   cmCathodeNgPnp2ndFwdBwd.monitoring.commandWorkPos := FALSE;
   cmCathodeNgPnp2ndFwdBwd.monitoring.goToHomePos := TRUE;
   cmCathodeNgPnp2ndFwdBwd.monitoring.goToWorkPos := FALSE;
   cmCathodeNgPnp2ndFwdBwd.monitoring.inHomePos := TRUE;
   cmCathodeNgPnp2ndFwdBwd.monitoring.inWorkPos := FALSE;
   cmCathodeNgPnp2ndFwdBwd.monitoring.reset := FALSE;
   cmCathodeNgPnp2ndFwdBwd.monitoring.enableManualCmds := FALSE;
   cmCathodeNgPnp2ndFwdBwd.monitoring.error := FALSE;
   cmCathodeNgPnp2ndFwdBwd.monitoring.interlockHomePos := TRUE;
   cmCathodeNgPnp2ndFwdBwd.monitoring.interlockWorkPos := TRUE;
   cmCathodeNgPnp2ndFwdBwd.monitoring.status := 16#7004;
   cmCathodeNgPnp2ndFwdBwd.monitoring.interlockWarningWorkPos := FALSE;
   cmCathodeNgPnp2ndFwdBwd.monitoring.interlockWarningHomePos := FALSE;
   cmCathodeNgPnp2ndFwdBwd.configuration.referenceDesignator := WSTRING#'CaNgPnp2ndFwdBwd';
   cmCathodeNgPnp2ndFwdBwd.configuration.monitoringLeavingFeedback := T#5S;
   cmCathodeNgPnp2ndFwdBwd.configuration.monitoringReachingFeedback := T#5S;
   cmCathodeNgPnp2ndFwdBwd.configuration.monitoringDiscrepancy := T#0MS;
   cmCathodeNgPnp2ndFwdBwd.configuration.setOutputHomeContinuously := TRUE;
   cmCathodeNgPnp2ndFwdBwd.configuration.setOutputWorkContinuously := TRUE;
   cmCathodeNgPnp2ndFwdBwd.configuration.disableHomeCommand := FALSE;
   cmCathodeNgPnp2ndFwdBwd.configuration.disableFeedbackHomePos := FALSE;
   cmCathodeNgPnp2ndFwdBwd.configuration.disableFeedbackWorkPos := FALSE;
   cmCathodeNgPnp2ndFwdBwd.configuration.disableAlarms := FALSE;
   cmCathodeNgPnp2ndFwdBwd.configuration.resetOutputsOnError := FALSE;
   cmCathodeNgPnp2ndFwdBwd.configuration.allwaysWaitOnReachingTime := FALSE;
   cmCathodeMaintenanceMovingFixFrontRearFwdBwd.commands.refreshConfiguration := FALSE;
   cmCathodeMaintenanceMovingFixFrontRearFwdBwd.commands.editConfiguration := FALSE;
   cmCathodeMaintenanceMovingFixFrontRearFwdBwd.commands.saveConfiguration := FALSE;
   cmCathodeMaintenanceMovingFixFrontRearFwdBwd.commands.reset := FALSE;
   cmCathodeMaintenanceMovingFixFrontRearFwdBwd.commands.commandHomePos := FALSE;
   cmCathodeMaintenanceMovingFixFrontRearFwdBwd.commands.commandWorkPos := FALSE;
   cmCathodeMaintenanceMovingFixFrontRearFwdBwd.monitoring.enable := TRUE;
   cmCathodeMaintenanceMovingFixFrontRearFwdBwd.monitoring.referenceDesignator := WSTRING#'MaintenanceFix';
   cmCathodeMaintenanceMovingFixFrontRearFwdBwd.monitoring.commandHomePos := FALSE;
   cmCathodeMaintenanceMovingFixFrontRearFwdBwd.monitoring.commandWorkPos := FALSE;
   cmCathodeMaintenanceMovingFixFrontRearFwdBwd.monitoring.goToHomePos := FALSE;
   cmCathodeMaintenanceMovingFixFrontRearFwdBwd.monitoring.goToWorkPos := FALSE;
   cmCathodeMaintenanceMovingFixFrontRearFwdBwd.monitoring.inHomePos := FALSE;
   cmCathodeMaintenanceMovingFixFrontRearFwdBwd.monitoring.inWorkPos := FALSE;
   cmCathodeMaintenanceMovingFixFrontRearFwdBwd.monitoring.reset := FALSE;
   cmCathodeMaintenanceMovingFixFrontRearFwdBwd.monitoring.enableManualCmds := FALSE;
   cmCathodeMaintenanceMovingFixFrontRearFwdBwd.monitoring.error := FALSE;
   cmCathodeMaintenanceMovingFixFrontRearFwdBwd.monitoring.interlockHomePos := TRUE;
   cmCathodeMaintenanceMovingFixFrontRearFwdBwd.monitoring.interlockWorkPos := TRUE;
   cmCathodeMaintenanceMovingFixFrontRearFwdBwd.monitoring.status := 16#7003;
   cmCathodeMaintenanceMovingFixFrontRearFwdBwd.monitoring.interlockWarningWorkPos := FALSE;
   cmCathodeMaintenanceMovingFixFrontRearFwdBwd.monitoring.interlockWarningHomePos := FALSE;
   cmCathodeMaintenanceMovingFixFrontRearFwdBwd.configuration.referenceDesignator := WSTRING#'CaMaintFixFrontRearFwdBwd';
   cmCathodeMaintenanceMovingFixFrontRearFwdBwd.configuration.monitoringLeavingFeedback := T#5S;
   cmCathodeMaintenanceMovingFixFrontRearFwdBwd.configuration.monitoringReachingFeedback := T#5S;
   cmCathodeMaintenanceMovingFixFrontRearFwdBwd.configuration.monitoringDiscrepancy := T#0MS;
   cmCathodeMaintenanceMovingFixFrontRearFwdBwd.configuration.setOutputHomeContinuously := TRUE;
   cmCathodeMaintenanceMovingFixFrontRearFwdBwd.configuration.setOutputWorkContinuously := TRUE;
   cmCathodeMaintenanceMovingFixFrontRearFwdBwd.configuration.disableHomeCommand := FALSE;
   cmCathodeMaintenanceMovingFixFrontRearFwdBwd.configuration.disableFeedbackHomePos := FALSE;
   cmCathodeMaintenanceMovingFixFrontRearFwdBwd.configuration.disableFeedbackWorkPos := FALSE;
   cmCathodeMaintenanceMovingFixFrontRearFwdBwd.configuration.disableAlarms := FALSE;
   cmCathodeMaintenanceMovingFixFrontRearFwdBwd.configuration.resetOutputsOnError := FALSE;
   cmCathodeMaintenanceMovingFixFrontRearFwdBwd.configuration.allwaysWaitOnReachingTime := FALSE;
   cmCathodeNgBoxLiftUpDown.commands.refreshConfiguration := FALSE;
   cmCathodeNgBoxLiftUpDown.commands.editConfiguration := FALSE;
   cmCathodeNgBoxLiftUpDown.commands.saveConfiguration := FALSE;
   cmCathodeNgBoxLiftUpDown.commands.reset := FALSE;
   cmCathodeNgBoxLiftUpDown.commands.commandHomePos := FALSE;
   cmCathodeNgBoxLiftUpDown.commands.commandWorkPos := FALSE;
   cmCathodeNgBoxLiftUpDown.monitoring.enable := TRUE;
   cmCathodeNgBoxLiftUpDown.monitoring.referenceDesignator := WSTRING#'NgBoxLiftUpDown';
   cmCathodeNgBoxLiftUpDown.monitoring.commandHomePos := FALSE;
   cmCathodeNgBoxLiftUpDown.monitoring.commandWorkPos := FALSE;
   cmCathodeNgBoxLiftUpDown.monitoring.goToHomePos := FALSE;
   cmCathodeNgBoxLiftUpDown.monitoring.goToWorkPos := TRUE;
   cmCathodeNgBoxLiftUpDown.monitoring.inHomePos := FALSE;
   cmCathodeNgBoxLiftUpDown.monitoring.inWorkPos := TRUE;
   cmCathodeNgBoxLiftUpDown.monitoring.reset := FALSE;
   cmCathodeNgBoxLiftUpDown.monitoring.enableManualCmds := FALSE;
   cmCathodeNgBoxLiftUpDown.monitoring.error := FALSE;
   cmCathodeNgBoxLiftUpDown.monitoring.interlockHomePos := TRUE;
   cmCathodeNgBoxLiftUpDown.monitoring.interlockWorkPos := TRUE;
   cmCathodeNgBoxLiftUpDown.monitoring.status := 16#7006;
   cmCathodeNgBoxLiftUpDown.monitoring.interlockWarningWorkPos := FALSE;
   cmCathodeNgBoxLiftUpDown.monitoring.interlockWarningHomePos := FALSE;
   cmCathodeNgBoxLiftUpDown.configuration.referenceDesignator := WSTRING#'CaNgBoxLiftUpDown';
   cmCathodeNgBoxLiftUpDown.configuration.monitoringLeavingFeedback := T#5S;
   cmCathodeNgBoxLiftUpDown.configuration.monitoringReachingFeedback := T#5S;
   cmCathodeNgBoxLiftUpDown.configuration.monitoringDiscrepancy := T#0MS;
   cmCathodeNgBoxLiftUpDown.configuration.setOutputHomeContinuously := TRUE;
   cmCathodeNgBoxLiftUpDown.configuration.setOutputWorkContinuously := TRUE;
   cmCathodeNgBoxLiftUpDown.configuration.disableHomeCommand := FALSE;
   cmCathodeNgBoxLiftUpDown.configuration.disableFeedbackHomePos := FALSE;
   cmCathodeNgBoxLiftUpDown.configuration.disableFeedbackWorkPos := FALSE;
   cmCathodeNgBoxLiftUpDown.configuration.disableAlarms := FALSE;
   cmCathodeNgBoxLiftUpDown.configuration.resetOutputsOnError := FALSE;
   cmCathodeNgBoxLiftUpDown.configuration.allwaysWaitOnReachingTime := FALSE;
   cmCathodeNgBoxLockUpDown.commands.refreshConfiguration := FALSE;
   cmCathodeNgBoxLockUpDown.commands.editConfiguration := FALSE;
   cmCathodeNgBoxLockUpDown.commands.saveConfiguration := FALSE;
   cmCathodeNgBoxLockUpDown.commands.reset := FALSE;
   cmCathodeNgBoxLockUpDown.commands.commandHomePos := FALSE;
   cmCathodeNgBoxLockUpDown.commands.commandWorkPos := FALSE;
   cmCathodeNgBoxLockUpDown.monitoring.enable := TRUE;
   cmCathodeNgBoxLockUpDown.monitoring.referenceDesignator := WSTRING#'NgBoxLockUpDown';
   cmCathodeNgBoxLockUpDown.monitoring.commandHomePos := FALSE;
   cmCathodeNgBoxLockUpDown.monitoring.commandWorkPos := FALSE;
   cmCathodeNgBoxLockUpDown.monitoring.goToHomePos := FALSE;
   cmCathodeNgBoxLockUpDown.monitoring.goToWorkPos := FALSE;
   cmCathodeNgBoxLockUpDown.monitoring.inHomePos := FALSE;
   cmCathodeNgBoxLockUpDown.monitoring.inWorkPos := FALSE;
   cmCathodeNgBoxLockUpDown.monitoring.reset := FALSE;
   cmCathodeNgBoxLockUpDown.monitoring.enableManualCmds := FALSE;
   cmCathodeNgBoxLockUpDown.monitoring.error := FALSE;
   cmCathodeNgBoxLockUpDown.monitoring.interlockHomePos := TRUE;
   cmCathodeNgBoxLockUpDown.monitoring.interlockWorkPos := FALSE;
   cmCathodeNgBoxLockUpDown.monitoring.status := 16#7101;
   cmCathodeNgBoxLockUpDown.monitoring.interlockWarningWorkPos := FALSE;
   cmCathodeNgBoxLockUpDown.monitoring.interlockWarningHomePos := FALSE;
   cmCathodeNgBoxLockUpDown.configuration.referenceDesignator := WSTRING#'CaNgBoxLockUpDown';
   cmCathodeNgBoxLockUpDown.configuration.monitoringLeavingFeedback := T#5S;
   cmCathodeNgBoxLockUpDown.configuration.monitoringReachingFeedback := T#5S;
   cmCathodeNgBoxLockUpDown.configuration.monitoringDiscrepancy := T#0MS;
   cmCathodeNgBoxLockUpDown.configuration.setOutputHomeContinuously := TRUE;
   cmCathodeNgBoxLockUpDown.configuration.setOutputWorkContinuously := TRUE;
   cmCathodeNgBoxLockUpDown.configuration.disableHomeCommand := FALSE;
   cmCathodeNgBoxLockUpDown.configuration.disableFeedbackHomePos := FALSE;
   cmCathodeNgBoxLockUpDown.configuration.disableFeedbackWorkPos := FALSE;
   cmCathodeNgBoxLockUpDown.configuration.disableAlarms := FALSE;
   cmCathodeNgBoxLockUpDown.configuration.resetOutputsOnError := FALSE;
   cmCathodeNgBoxLockUpDown.configuration.allwaysWaitOnReachingTime := FALSE;
   cmCathodeNgPnpVaccum.commands.refreshConfiguration := FALSE;
   cmCathodeNgPnpVaccum.commands.editConfiguration := FALSE;
   cmCathodeNgPnpVaccum.commands.saveConfiguration := FALSE;
   cmCathodeNgPnpVaccum.commands.reset := FALSE;
   cmCathodeNgPnpVaccum.commands.commandHomePos := FALSE;
   cmCathodeNgPnpVaccum.commands.commandWorkPos := FALSE;
   cmCathodeNgPnpVaccum.monitoring.enable := TRUE;
   cmCathodeNgPnpVaccum.monitoring.referenceDesignator := WSTRING#'NgPnpVaccum';
   cmCathodeNgPnpVaccum.monitoring.commandHomePos := FALSE;
   cmCathodeNgPnpVaccum.monitoring.commandWorkPos := FALSE;
   cmCathodeNgPnpVaccum.monitoring.goToHomePos := FALSE;
   cmCathodeNgPnpVaccum.monitoring.goToWorkPos := FALSE;
   cmCathodeNgPnpVaccum.monitoring.inHomePos := TRUE;
   cmCathodeNgPnpVaccum.monitoring.inWorkPos := FALSE;
   cmCathodeNgPnpVaccum.monitoring.reset := FALSE;
   cmCathodeNgPnpVaccum.monitoring.enableManualCmds := FALSE;
   cmCathodeNgPnpVaccum.monitoring.error := FALSE;
   cmCathodeNgPnpVaccum.monitoring.interlockHomePos := TRUE;
   cmCathodeNgPnpVaccum.monitoring.interlockWorkPos := TRUE;
   cmCathodeNgPnpVaccum.monitoring.status := 16#7003;
   cmCathodeNgPnpVaccum.monitoring.interlockWarningWorkPos := FALSE;
   cmCathodeNgPnpVaccum.monitoring.interlockWarningHomePos := FALSE;
   cmCathodeNgPnpVaccum.configuration.referenceDesignator := WSTRING#'CaNgPnpVaccum';
   cmCathodeNgPnpVaccum.configuration.monitoringLeavingFeedback := T#5S;
   cmCathodeNgPnpVaccum.configuration.monitoringReachingFeedback := T#5S;
   cmCathodeNgPnpVaccum.configuration.monitoringDiscrepancy := T#0MS;
   cmCathodeNgPnpVaccum.configuration.setOutputHomeContinuously := TRUE;
   cmCathodeNgPnpVaccum.configuration.setOutputWorkContinuously := TRUE;
   cmCathodeNgPnpVaccum.configuration.disableHomeCommand := FALSE;
   cmCathodeNgPnpVaccum.configuration.disableFeedbackHomePos := FALSE;
   cmCathodeNgPnpVaccum.configuration.disableFeedbackWorkPos := FALSE;
   cmCathodeNgPnpVaccum.configuration.disableAlarms := FALSE;
   cmCathodeNgPnpVaccum.configuration.resetOutputsOnError := FALSE;
   cmCathodeNgPnpVaccum.configuration.allwaysWaitOnReachingTime := FALSE;
   cmCathodeConveyorCoverFwdBwd.commands.refreshConfiguration := FALSE;
   cmCathodeConveyorCoverFwdBwd.commands.editConfiguration := FALSE;
   cmCathodeConveyorCoverFwdBwd.commands.saveConfiguration := FALSE;
   cmCathodeConveyorCoverFwdBwd.commands.reset := FALSE;
   cmCathodeConveyorCoverFwdBwd.commands.commandHomePos := FALSE;
   cmCathodeConveyorCoverFwdBwd.commands.commandWorkPos := FALSE;
   cmCathodeConveyorCoverFwdBwd.monitoring.enable := TRUE;
   cmCathodeConveyorCoverFwdBwd.monitoring.referenceDesignator := WSTRING#'ConveyorCoverFwdBwd';
   cmCathodeConveyorCoverFwdBwd.monitoring.commandHomePos := FALSE;
   cmCathodeConveyorCoverFwdBwd.monitoring.commandWorkPos := FALSE;
   cmCathodeConveyorCoverFwdBwd.monitoring.goToHomePos := FALSE;
   cmCathodeConveyorCoverFwdBwd.monitoring.goToWorkPos := FALSE;
   cmCathodeConveyorCoverFwdBwd.monitoring.inHomePos := FALSE;
   cmCathodeConveyorCoverFwdBwd.monitoring.inWorkPos := FALSE;
   cmCathodeConveyorCoverFwdBwd.monitoring.reset := FALSE;
   cmCathodeConveyorCoverFwdBwd.monitoring.enableManualCmds := FALSE;
   cmCathodeConveyorCoverFwdBwd.monitoring.error := FALSE;
   cmCathodeConveyorCoverFwdBwd.monitoring.interlockHomePos := TRUE;
   cmCathodeConveyorCoverFwdBwd.monitoring.interlockWorkPos := TRUE;
   cmCathodeConveyorCoverFwdBwd.monitoring.status := 16#7003;
   cmCathodeConveyorCoverFwdBwd.monitoring.interlockWarningWorkPos := FALSE;
   cmCathodeConveyorCoverFwdBwd.monitoring.interlockWarningHomePos := FALSE;
   cmCathodeConveyorCoverFwdBwd.configuration.referenceDesignator := WSTRING#'CaConvCoverFwdBwd';
   cmCathodeConveyorCoverFwdBwd.configuration.monitoringLeavingFeedback := T#5S;
   cmCathodeConveyorCoverFwdBwd.configuration.monitoringReachingFeedback := T#5S;
   cmCathodeConveyorCoverFwdBwd.configuration.monitoringDiscrepancy := T#0MS;
   cmCathodeConveyorCoverFwdBwd.configuration.setOutputHomeContinuously := TRUE;
   cmCathodeConveyorCoverFwdBwd.configuration.setOutputWorkContinuously := TRUE;
   cmCathodeConveyorCoverFwdBwd.configuration.disableHomeCommand := FALSE;
   cmCathodeConveyorCoverFwdBwd.configuration.disableFeedbackHomePos := FALSE;
   cmCathodeConveyorCoverFwdBwd.configuration.disableFeedbackWorkPos := FALSE;
   cmCathodeConveyorCoverFwdBwd.configuration.disableAlarms := FALSE;
   cmCathodeConveyorCoverFwdBwd.configuration.resetOutputsOnError := FALSE;
   cmCathodeConveyorCoverFwdBwd.configuration.allwaysWaitOnReachingTime := FALSE;
   cmCathodeConveyorPickUpBlower.commands.refreshConfiguration := FALSE;
   cmCathodeConveyorPickUpBlower.commands.editConfiguration := FALSE;
   cmCathodeConveyorPickUpBlower.commands.saveConfiguration := FALSE;
   cmCathodeConveyorPickUpBlower.commands.reset := FALSE;
   cmCathodeConveyorPickUpBlower.commands.commandHomePos := FALSE;
   cmCathodeConveyorPickUpBlower.commands.commandWorkPos := FALSE;
   cmCathodeConveyorPickUpBlower.monitoring.enable := TRUE;
   cmCathodeConveyorPickUpBlower.monitoring.referenceDesignator := WSTRING#'ConveyorPickUpBlower';
   cmCathodeConveyorPickUpBlower.monitoring.commandHomePos := FALSE;
   cmCathodeConveyorPickUpBlower.monitoring.commandWorkPos := FALSE;
   cmCathodeConveyorPickUpBlower.monitoring.goToHomePos := FALSE;
   cmCathodeConveyorPickUpBlower.monitoring.goToWorkPos := TRUE;
   cmCathodeConveyorPickUpBlower.monitoring.inHomePos := FALSE;
   cmCathodeConveyorPickUpBlower.monitoring.inWorkPos := TRUE;
   cmCathodeConveyorPickUpBlower.monitoring.reset := FALSE;
   cmCathodeConveyorPickUpBlower.monitoring.enableManualCmds := FALSE;
   cmCathodeConveyorPickUpBlower.monitoring.error := FALSE;
   cmCathodeConveyorPickUpBlower.monitoring.interlockHomePos := TRUE;
   cmCathodeConveyorPickUpBlower.monitoring.interlockWorkPos := TRUE;
   cmCathodeConveyorPickUpBlower.monitoring.status := 16#7006;
   cmCathodeConveyorPickUpBlower.monitoring.interlockWarningWorkPos := FALSE;
   cmCathodeConveyorPickUpBlower.monitoring.interlockWarningHomePos := FALSE;
   cmCathodeConveyorPickUpBlower.configuration.referenceDesignator := WSTRING#'CaConvPickUpBlower';
   cmCathodeConveyorPickUpBlower.configuration.monitoringLeavingFeedback := T#5S;
   cmCathodeConveyorPickUpBlower.configuration.monitoringReachingFeedback := T#5S;
   cmCathodeConveyorPickUpBlower.configuration.monitoringDiscrepancy := T#0MS;
   cmCathodeConveyorPickUpBlower.configuration.setOutputHomeContinuously := TRUE;
   cmCathodeConveyorPickUpBlower.configuration.setOutputWorkContinuously := TRUE;
   cmCathodeConveyorPickUpBlower.configuration.disableHomeCommand := FALSE;
   cmCathodeConveyorPickUpBlower.configuration.disableFeedbackHomePos := FALSE;
   cmCathodeConveyorPickUpBlower.configuration.disableFeedbackWorkPos := FALSE;
   cmCathodeConveyorPickUpBlower.configuration.disableAlarms := FALSE;
   cmCathodeConveyorPickUpBlower.configuration.resetOutputsOnError := FALSE;
   cmCathodeConveyorPickUpBlower.configuration.allwaysWaitOnReachingTime := FALSE;
   cmAlignVisionControllerInterface.commands.stepStart := FALSE;
   cmAlignVisionControllerInterface.commands.errorAck := FALSE;
   cmAlignVisionControllerInterface.commands.dataDelete := FALSE;
   cmAlignVisionControllerInterface.monitoring.profinetInput.cmdResultStatus.cmdComplete := FALSE;
   cmAlignVisionControllerInterface.monitoring.profinetInput.cmdResultStatus.cmdError := FALSE;
   cmAlignVisionControllerInterface.monitoring.profinetInput.cmdResultStatus.cmdReady := FALSE;
   cmAlignVisionControllerInterface.monitoring.profinetInput.cmdResultStatus.resultReady := FALSE;
   cmAlignVisionControllerInterface.monitoring.profinetInput.cmdResultStatus.resultOR := FALSE;
   cmAlignVisionControllerInterface.monitoring.profinetInput.cmdResultStatus.reserved0 := FALSE;
   cmAlignVisionControllerInterface.monitoring.profinetInput.cmdResultStatus.reserved1 := FALSE;
   cmAlignVisionControllerInterface.monitoring.profinetInput.cmdResultStatus.reserved2 := FALSE;
   cmAlignVisionControllerInterface.monitoring.profinetInput.trgReadyStatus.trg1Ready := FALSE;
   cmAlignVisionControllerInterface.monitoring.profinetInput.trgReadyStatus.trg2Ready := FALSE;
   cmAlignVisionControllerInterface.monitoring.profinetInput.trgReadyStatus.trg3Ready := FALSE;
   cmAlignVisionControllerInterface.monitoring.profinetInput.trgReadyStatus.trg4Ready := FALSE;
   cmAlignVisionControllerInterface.monitoring.profinetInput.trgReadyStatus.reserved0 := FALSE;
   cmAlignVisionControllerInterface.monitoring.profinetInput.trgReadyStatus.reserved1 := FALSE;
   cmAlignVisionControllerInterface.monitoring.profinetInput.trgReadyStatus.reserved2 := FALSE;
   cmAlignVisionControllerInterface.monitoring.profinetInput.trgReadyStatus.reserved3 := FALSE;
   cmAlignVisionControllerInterface.monitoring.profinetInput.trgAckStatus.trg1Ack := FALSE;
   cmAlignVisionControllerInterface.monitoring.profinetInput.trgAckStatus.trg2Ack := FALSE;
   cmAlignVisionControllerInterface.monitoring.profinetInput.trgAckStatus.trg3Ack := FALSE;
   cmAlignVisionControllerInterface.monitoring.profinetInput.trgAckStatus.trg4Ack := FALSE;
   cmAlignVisionControllerInterface.monitoring.profinetInput.trgAckStatus.reserved0 := FALSE;
   cmAlignVisionControllerInterface.monitoring.profinetInput.trgAckStatus.reserved1 := FALSE;
   cmAlignVisionControllerInterface.monitoring.profinetInput.trgAckStatus.reserved2 := FALSE;
   cmAlignVisionControllerInterface.monitoring.profinetInput.trgAckStatus.reserved3 := FALSE;
   cmAlignVisionControllerInterface.monitoring.profinetInput.miscellaneousStatus.busy := FALSE;
   cmAlignVisionControllerInterface.monitoring.profinetInput.miscellaneousStatus.err0Status := FALSE;
   cmAlignVisionControllerInterface.monitoring.profinetInput.miscellaneousStatus.err1Status := FALSE;
   cmAlignVisionControllerInterface.monitoring.profinetInput.miscellaneousStatus.remoteReady := FALSE;
   cmAlignVisionControllerInterface.monitoring.profinetInput.miscellaneousStatus.reserved0 := FALSE;
   cmAlignVisionControllerInterface.monitoring.profinetInput.miscellaneousStatus.reserved1 := FALSE;
   cmAlignVisionControllerInterface.monitoring.profinetInput.miscellaneousStatus.reserved2 := FALSE;
   cmAlignVisionControllerInterface.monitoring.profinetInput.miscellaneousStatus.reserved3 := FALSE;
   cmAlignVisionControllerInterface.monitoring.profinetInput.assignableStatus.assignable_0 := FALSE;
   cmAlignVisionControllerInterface.monitoring.profinetInput.assignableStatus.assignable_1 := FALSE;
   cmAlignVisionControllerInterface.monitoring.profinetInput.assignableStatus.assignable_2 := FALSE;
   cmAlignVisionControllerInterface.monitoring.profinetInput.assignableStatus.assignable_3 := FALSE;
   cmAlignVisionControllerInterface.monitoring.profinetInput.assignableStatus.assignable_4 := FALSE;
   cmAlignVisionControllerInterface.monitoring.profinetInput.assignableStatus.assignable_5 := FALSE;
   cmAlignVisionControllerInterface.monitoring.profinetInput.assignableStatus.assignable_6 := FALSE;
   cmAlignVisionControllerInterface.monitoring.profinetInput.assignableStatus.assignable_7 := FALSE;
   cmAlignVisionControllerInterface.monitoring.profinetInput.assignableStatus.assignable_8 := FALSE;
   cmAlignVisionControllerInterface.monitoring.profinetInput.assignableStatus.assignable_9 := FALSE;
   cmAlignVisionControllerInterface.monitoring.profinetInput.assignableStatus.assignable_10 := FALSE;
   cmAlignVisionControllerInterface.monitoring.profinetInput.assignableStatus.assignable_11 := FALSE;
   cmAlignVisionControllerInterface.monitoring.profinetInput.assignableStatus.assignable_12 := FALSE;
   cmAlignVisionControllerInterface.monitoring.profinetInput.assignableStatus.assignable_13 := FALSE;
   cmAlignVisionControllerInterface.monitoring.profinetInput.assignableStatus.assignable_14 := FALSE;
   cmAlignVisionControllerInterface.monitoring.profinetInput.assignableStatus.assignable_15 := FALSE;
   cmAlignVisionControllerInterface.monitoring.profinetInput.assignableStatus.assignable_16 := FALSE;
   cmAlignVisionControllerInterface.monitoring.profinetInput.assignableStatus.assignable_17 := FALSE;
   cmAlignVisionControllerInterface.monitoring.profinetInput.assignableStatus.assignable_18 := FALSE;
   cmAlignVisionControllerInterface.monitoring.profinetInput.assignableStatus.assignable_19 := FALSE;
   cmAlignVisionControllerInterface.monitoring.profinetInput.assignableStatus.assignable_20 := FALSE;
   cmAlignVisionControllerInterface.monitoring.profinetInput.assignableStatus.assignable_21 := FALSE;
   cmAlignVisionControllerInterface.monitoring.profinetInput.assignableStatus.assignable_22 := FALSE;
   cmAlignVisionControllerInterface.monitoring.profinetInput.assignableStatus.assignable_23 := FALSE;
   cmAlignVisionControllerInterface.monitoring.profinetInput.assignableStatus.assignable_24 := FALSE;
   cmAlignVisionControllerInterface.monitoring.profinetInput.assignableStatus.assignable_25 := FALSE;
   cmAlignVisionControllerInterface.monitoring.profinetInput.assignableStatus.assignable_26 := FALSE;
   cmAlignVisionControllerInterface.monitoring.profinetInput.assignableStatus.assignable_27 := FALSE;
   cmAlignVisionControllerInterface.monitoring.profinetInput.assignableStatus.assignable_28 := FALSE;
   cmAlignVisionControllerInterface.monitoring.profinetInput.assignableStatus.assignable_29 := FALSE;
   cmAlignVisionControllerInterface.monitoring.profinetInput.assignableStatus.assignable_30 := FALSE;
   cmAlignVisionControllerInterface.monitoring.profinetInput.assignableStatus.assignable_31 := FALSE;
   cmAlignVisionControllerInterface.monitoring.profinetInput.resultData248Byte_1.error0Code := 0;
   cmAlignVisionControllerInterface.monitoring.profinetInput.resultData248Byte_1.error1Code := 0;
   cmAlignVisionControllerInterface.monitoring.profinetInput.resultData248Byte_1.reserved12 := 0;
   cmAlignVisionControllerInterface.monitoring.profinetInput.resultData248Byte_1.totalCount := 0;
   cmAlignVisionControllerInterface.monitoring.profinetInput.resultData248Byte_1.commandResult := 0;
   cmAlignVisionControllerInterface.monitoring.profinetInput.resultData248Byte_1.commandData[0..23] := 0;
   cmAlignVisionControllerInterface.monitoring.profinetInput.resultData248Byte_1.resultData[0..33] := 0;
   cmAlignVisionControllerInterface.monitoring.profinetInput.resultData248Byte_2[0..61] := 0;
   cmAlignVisionControllerInterface.monitoring.profinetInput.resultData248Byte_3[0..61] := 0;
   cmAlignVisionControllerInterface.monitoring.profinetInput.resultData248Byte_4[0..61] := 0;
   cmAlignVisionControllerInterface.monitoring.profinetInput.resultData248Byte_5[0..61] := 0;
   cmAlignVisionControllerInterface.monitoring.profinetOutput.cmdResultControl.cmdRequest := FALSE;
   cmAlignVisionControllerInterface.monitoring.profinetOutput.cmdResultControl.inDataFbSyncInhibit := FALSE;
   cmAlignVisionControllerInterface.monitoring.profinetOutput.cmdResultControl.reserved := FALSE;
   cmAlignVisionControllerInterface.monitoring.profinetOutput.cmdResultControl.resultAck := FALSE;
   cmAlignVisionControllerInterface.monitoring.profinetOutput.cmdResultControl.err0ResetRequest := FALSE;
   cmAlignVisionControllerInterface.monitoring.profinetOutput.cmdResultControl.err1ResetRequest := FALSE;
   cmAlignVisionControllerInterface.monitoring.profinetOutput.cmdResultControl.reserved0 := FALSE;
   cmAlignVisionControllerInterface.monitoring.profinetOutput.cmdResultControl.reserved1 := FALSE;
   cmAlignVisionControllerInterface.monitoring.profinetOutput.trgControl.trg1 := FALSE;
   cmAlignVisionControllerInterface.monitoring.profinetOutput.trgControl.trg2 := FALSE;
   cmAlignVisionControllerInterface.monitoring.profinetOutput.trgControl.trg3 := FALSE;
   cmAlignVisionControllerInterface.monitoring.profinetOutput.trgControl.trg4 := FALSE;
   cmAlignVisionControllerInterface.monitoring.profinetOutput.trgControl.reserved0 := FALSE;
   cmAlignVisionControllerInterface.monitoring.profinetOutput.trgControl.reserved1 := FALSE;
   cmAlignVisionControllerInterface.monitoring.profinetOutput.trgControl.reserved2 := FALSE;
   cmAlignVisionControllerInterface.monitoring.profinetOutput.trgControl.reserved3 := FALSE;
   cmAlignVisionControllerInterface.monitoring.profinetOutput.miscellaneousControl.reset := FALSE;
   cmAlignVisionControllerInterface.monitoring.profinetOutput.miscellaneousControl.ext := FALSE;
   cmAlignVisionControllerInterface.monitoring.profinetOutput.miscellaneousControl.test := FALSE;
   cmAlignVisionControllerInterface.monitoring.profinetOutput.miscellaneousControl.reserved0 := FALSE;
   cmAlignVisionControllerInterface.monitoring.profinetOutput.miscellaneousControl.reserved1 := FALSE;
   cmAlignVisionControllerInterface.monitoring.profinetOutput.miscellaneousControl.reserved2 := FALSE;
   cmAlignVisionControllerInterface.monitoring.profinetOutput.miscellaneousControl.reserved3 := FALSE;
   cmAlignVisionControllerInterface.monitoring.profinetOutput.miscellaneousControl.reserved4 := FALSE;
   cmAlignVisionControllerInterface.monitoring.profinetOutput.reservedControl.reserved0 := FALSE;
   cmAlignVisionControllerInterface.monitoring.profinetOutput.reservedControl.reserved1 := FALSE;
   cmAlignVisionControllerInterface.monitoring.profinetOutput.reservedControl.reserved2 := FALSE;
   cmAlignVisionControllerInterface.monitoring.profinetOutput.reservedControl.reserved3 := FALSE;
   cmAlignVisionControllerInterface.monitoring.profinetOutput.reservedControl.reserved4 := FALSE;
   cmAlignVisionControllerInterface.monitoring.profinetOutput.reservedControl.reserved5 := FALSE;
   cmAlignVisionControllerInterface.monitoring.profinetOutput.reservedControl.reserved6 := FALSE;
   cmAlignVisionControllerInterface.monitoring.profinetOutput.reservedControl.reserved7 := FALSE;
   cmAlignVisionControllerInterface.monitoring.profinetOutput.assignableControl.assignable_0 := FALSE;
   cmAlignVisionControllerInterface.monitoring.profinetOutput.assignableControl.assignable_1 := FALSE;
   cmAlignVisionControllerInterface.monitoring.profinetOutput.assignableControl.assignable_2 := FALSE;
   cmAlignVisionControllerInterface.monitoring.profinetOutput.assignableControl.assignable_3 := FALSE;
   cmAlignVisionControllerInterface.monitoring.profinetOutput.assignableControl.assignable_4 := FALSE;
   cmAlignVisionControllerInterface.monitoring.profinetOutput.assignableControl.assignable_5 := FALSE;
   cmAlignVisionControllerInterface.monitoring.profinetOutput.assignableControl.assignable_6 := FALSE;
   cmAlignVisionControllerInterface.monitoring.profinetOutput.assignableControl.assignable_7 := FALSE;
   cmAlignVisionControllerInterface.monitoring.profinetOutput.assignableControl.assignable_8 := FALSE;
   cmAlignVisionControllerInterface.monitoring.profinetOutput.assignableControl.assignable_9 := FALSE;
   cmAlignVisionControllerInterface.monitoring.profinetOutput.assignableControl.assignable_10 := FALSE;
   cmAlignVisionControllerInterface.monitoring.profinetOutput.assignableControl.assignable_11 := FALSE;
   cmAlignVisionControllerInterface.monitoring.profinetOutput.assignableControl.assignable_12 := FALSE;
   cmAlignVisionControllerInterface.monitoring.profinetOutput.assignableControl.assignable_13 := FALSE;
   cmAlignVisionControllerInterface.monitoring.profinetOutput.assignableControl.assignable_14 := FALSE;
   cmAlignVisionControllerInterface.monitoring.profinetOutput.assignableControl.assignable_15 := FALSE;
   cmAlignVisionControllerInterface.monitoring.profinetOutput.assignableControl.assignable_16 := FALSE;
   cmAlignVisionControllerInterface.monitoring.profinetOutput.assignableControl.assignable_17 := FALSE;
   cmAlignVisionControllerInterface.monitoring.profinetOutput.assignableControl.assignable_18 := FALSE;
   cmAlignVisionControllerInterface.monitoring.profinetOutput.assignableControl.assignable_19 := FALSE;
   cmAlignVisionControllerInterface.monitoring.profinetOutput.assignableControl.assignable_20 := FALSE;
   cmAlignVisionControllerInterface.monitoring.profinetOutput.assignableControl.assignable_21 := FALSE;
   cmAlignVisionControllerInterface.monitoring.profinetOutput.assignableControl.assignable_22 := FALSE;
   cmAlignVisionControllerInterface.monitoring.profinetOutput.assignableControl.assignable_23 := FALSE;
   cmAlignVisionControllerInterface.monitoring.profinetOutput.assignableControl.assignable_24 := FALSE;
   cmAlignVisionControllerInterface.monitoring.profinetOutput.assignableControl.assignable_25 := FALSE;
   cmAlignVisionControllerInterface.monitoring.profinetOutput.assignableControl.assignable_26 := FALSE;
   cmAlignVisionControllerInterface.monitoring.profinetOutput.assignableControl.assignable_27 := FALSE;
   cmAlignVisionControllerInterface.monitoring.profinetOutput.assignableControl.assignable_28 := FALSE;
   cmAlignVisionControllerInterface.monitoring.profinetOutput.assignableControl.assignable_29 := FALSE;
   cmAlignVisionControllerInterface.monitoring.profinetOutput.assignableControl.assignable_30 := FALSE;
   cmAlignVisionControllerInterface.monitoring.profinetOutput.assignableControl.assignable_31 := FALSE;
   cmAlignVisionControllerInterface.monitoring.profinetOutput.parameterData248Byte_1.reversed0 := 0;
   cmAlignVisionControllerInterface.monitoring.profinetOutput.parameterData248Byte_1.reserved1 := 0;
   cmAlignVisionControllerInterface.monitoring.profinetOutput.parameterData248Byte_1.commandNumber := 0;
   cmAlignVisionControllerInterface.monitoring.profinetOutput.parameterData248Byte_1.cmdParameter[0..15] := 0;
   cmAlignVisionControllerInterface.monitoring.profinetOutput.parameterData248Byte_1.inDataFieldbus[0..42] := 0;
   cmAlignVisionControllerInterface.monitoring.profinetOutput.parameterData248Byte_2[0..61] := 0;
   cmAlignVisionControllerInterface.monitoring.profinetOutput.parameterData248Byte_3[0..61] := 0;
   cmAlignVisionControllerInterface.monitoring.profinetOutput.parameterData248Byte_4[0..61] := 0;
   cmAlignVisionControllerInterface.monitoring.profinetOutput.parameterData248Byte_5[0..61] := 0;
   cmAlignVisionControllerInterface.monitoring.resultOK := FALSE;
   cmAlignVisionControllerInterface.monitoring.resultNG := FALSE;
   cmAlignVisionControllerInterface.monitoring.resultBusy := FALSE;
   cmAlignVisionControllerInterface.monitoring.resultComplete := FALSE;
   cmAlignVisionControllerInterface.monitoring.resultData.resultData136Byte_1[0..33] := 0;
   cmAlignVisionControllerInterface.monitoring.resultData.resultData248Byte_2[0..61] := 0;
   cmAlignVisionControllerInterface.monitoring.resultData.resultData248Byte_3[0..61] := 0;
   cmAlignVisionControllerInterface.monitoring.resultData.resultData248Byte_4[0..61] := 0;
   cmAlignVisionControllerInterface.monitoring.resultData.resultData248Byte_5[0..61] := 0;
   cmAlignVisionControllerInterface.monitoring.error := FALSE;
   cmAlignVisionControllerInterface.monitoring.status := 16#0000;
   cmAlignVisionControllerInterface.configuration.hwID.cmdResultStatusID := 0;
   cmAlignVisionControllerInterface.configuration.hwID.trgReadyStatusID := 0;
   cmAlignVisionControllerInterface.configuration.hwID.trgAckStatusID := 0;
   cmAlignVisionControllerInterface.configuration.hwID.miscellaneousStatusID := 0;
   cmAlignVisionControllerInterface.configuration.hwID.assignableStatusID := 0;
   cmAlignVisionControllerInterface.configuration.hwID.resultData248ByteID_1 := 0;
   cmAlignVisionControllerInterface.configuration.hwID.resultData248ByteID_2 := 0;
   cmAlignVisionControllerInterface.configuration.hwID.resultData248ByteID_3 := 0;
   cmAlignVisionControllerInterface.configuration.hwID.resultData248ByteID_4 := 0;
   cmAlignVisionControllerInterface.configuration.hwID.resultData248ByteID_5 := 0;
   cmAlignVisionControllerInterface.configuration.hwID.cmdResultControlID := 0;
   cmAlignVisionControllerInterface.configuration.hwID.trgControlID := 0;
   cmAlignVisionControllerInterface.configuration.hwID.miscellaneousControlID := 0;
   cmAlignVisionControllerInterface.configuration.hwID.reservedControlID := 0;
   cmAlignVisionControllerInterface.configuration.hwID.assignableControlID := 0;
   cmAlignVisionControllerInterface.configuration.hwID.parameterData248ByteID_1 := 0;
   cmAlignVisionControllerInterface.configuration.hwID.parameterData248ByteID_2 := 0;
   cmAlignVisionControllerInterface.configuration.hwID.parameterData248ByteID_3 := 0;
   cmAlignVisionControllerInterface.configuration.hwID.parameterData248ByteID_4 := 0;
   cmAlignVisionControllerInterface.configuration.hwID.parameterData248ByteID_5 := 0;
   cmAlignVisionControllerInterface.configuration.referenceDesignator := WSTRING#'';
   cmAlignVisionControllerInterface.configuration.disableAlarms := FALSE;
   cmAlignVisionControllerInterface.configuration.trigger1Use := FALSE;
   cmAlignVisionControllerInterface.configuration.trigger2Use := FALSE;
   cmAlignVisionControllerInterface.configuration.trigger3Use := FALSE;
   cmAlignVisionControllerInterface.configuration.trigger4Use := FALSE;
   cmAlignVisionControllerInterface.configuration.triggertime := T#0MS;
   cmAlignVisionControllerInterface.configuration.cycleTime := T#0MS;
   cmAlignVisionControllerInterface.configuration.DataConfig.cmdResultControl.cmdRequest := FALSE;
   cmAlignVisionControllerInterface.configuration.DataConfig.cmdResultControl.inDataFbSyncInhibit := FALSE;
   cmAlignVisionControllerInterface.configuration.DataConfig.cmdResultControl.reserved := FALSE;
   cmAlignVisionControllerInterface.configuration.DataConfig.cmdResultControl.resultAck := FALSE;
   cmAlignVisionControllerInterface.configuration.DataConfig.cmdResultControl.err0ResetRequest := FALSE;
   cmAlignVisionControllerInterface.configuration.DataConfig.cmdResultControl.err1ResetRequest := FALSE;
   cmAlignVisionControllerInterface.configuration.DataConfig.cmdResultControl.reserved0 := FALSE;
   cmAlignVisionControllerInterface.configuration.DataConfig.cmdResultControl.reserved1 := FALSE;
   cmAlignVisionControllerInterface.configuration.DataConfig.trgControl.trg1 := FALSE;
   cmAlignVisionControllerInterface.configuration.DataConfig.trgControl.trg2 := FALSE;
   cmAlignVisionControllerInterface.configuration.DataConfig.trgControl.trg3 := FALSE;
   cmAlignVisionControllerInterface.configuration.DataConfig.trgControl.trg4 := FALSE;
   cmAlignVisionControllerInterface.configuration.DataConfig.trgControl.reserved0 := FALSE;
   cmAlignVisionControllerInterface.configuration.DataConfig.trgControl.reserved1 := FALSE;
   cmAlignVisionControllerInterface.configuration.DataConfig.trgControl.reserved2 := FALSE;
   cmAlignVisionControllerInterface.configuration.DataConfig.trgControl.reserved3 := FALSE;
   cmAlignVisionControllerInterface.configuration.DataConfig.miscellaneousControl.reset := FALSE;
   cmAlignVisionControllerInterface.configuration.DataConfig.miscellaneousControl.ext := FALSE;
   cmAlignVisionControllerInterface.configuration.DataConfig.miscellaneousControl.test := FALSE;
   cmAlignVisionControllerInterface.configuration.DataConfig.miscellaneousControl.reserved0 := FALSE;
   cmAlignVisionControllerInterface.configuration.DataConfig.miscellaneousControl.reserved1 := FALSE;
   cmAlignVisionControllerInterface.configuration.DataConfig.miscellaneousControl.reserved2 := FALSE;
   cmAlignVisionControllerInterface.configuration.DataConfig.miscellaneousControl.reserved3 := FALSE;
   cmAlignVisionControllerInterface.configuration.DataConfig.miscellaneousControl.reserved4 := FALSE;
   cmAlignVisionControllerInterface.configuration.DataConfig.reservedControl.reserved0 := FALSE;
   cmAlignVisionControllerInterface.configuration.DataConfig.reservedControl.reserved1 := FALSE;
   cmAlignVisionControllerInterface.configuration.DataConfig.reservedControl.reserved2 := FALSE;
   cmAlignVisionControllerInterface.configuration.DataConfig.reservedControl.reserved3 := FALSE;
   cmAlignVisionControllerInterface.configuration.DataConfig.reservedControl.reserved4 := FALSE;
   cmAlignVisionControllerInterface.configuration.DataConfig.reservedControl.reserved5 := FALSE;
   cmAlignVisionControllerInterface.configuration.DataConfig.reservedControl.reserved6 := FALSE;
   cmAlignVisionControllerInterface.configuration.DataConfig.reservedControl.reserved7 := FALSE;
   cmAlignVisionControllerInterface.configuration.DataConfig.assignableControl.assignable_0 := FALSE;
   cmAlignVisionControllerInterface.configuration.DataConfig.assignableControl.assignable_1 := FALSE;
   cmAlignVisionControllerInterface.configuration.DataConfig.assignableControl.assignable_2 := FALSE;
   cmAlignVisionControllerInterface.configuration.DataConfig.assignableControl.assignable_3 := FALSE;
   cmAlignVisionControllerInterface.configuration.DataConfig.assignableControl.assignable_4 := FALSE;
   cmAlignVisionControllerInterface.configuration.DataConfig.assignableControl.assignable_5 := FALSE;
   cmAlignVisionControllerInterface.configuration.DataConfig.assignableControl.assignable_6 := FALSE;
   cmAlignVisionControllerInterface.configuration.DataConfig.assignableControl.assignable_7 := FALSE;
   cmAlignVisionControllerInterface.configuration.DataConfig.assignableControl.assignable_8 := FALSE;
   cmAlignVisionControllerInterface.configuration.DataConfig.assignableControl.assignable_9 := FALSE;
   cmAlignVisionControllerInterface.configuration.DataConfig.assignableControl.assignable_10 := FALSE;
   cmAlignVisionControllerInterface.configuration.DataConfig.assignableControl.assignable_11 := FALSE;
   cmAlignVisionControllerInterface.configuration.DataConfig.assignableControl.assignable_12 := FALSE;
   cmAlignVisionControllerInterface.configuration.DataConfig.assignableControl.assignable_13 := FALSE;
   cmAlignVisionControllerInterface.configuration.DataConfig.assignableControl.assignable_14 := FALSE;
   cmAlignVisionControllerInterface.configuration.DataConfig.assignableControl.assignable_15 := FALSE;
   cmAlignVisionControllerInterface.configuration.DataConfig.assignableControl.assignable_16 := FALSE;
   cmAlignVisionControllerInterface.configuration.DataConfig.assignableControl.assignable_17 := FALSE;
   cmAlignVisionControllerInterface.configuration.DataConfig.assignableControl.assignable_18 := FALSE;
   cmAlignVisionControllerInterface.configuration.DataConfig.assignableControl.assignable_19 := FALSE;
   cmAlignVisionControllerInterface.configuration.DataConfig.assignableControl.assignable_20 := FALSE;
   cmAlignVisionControllerInterface.configuration.DataConfig.assignableControl.assignable_21 := FALSE;
   cmAlignVisionControllerInterface.configuration.DataConfig.assignableControl.assignable_22 := FALSE;
   cmAlignVisionControllerInterface.configuration.DataConfig.assignableControl.assignable_23 := FALSE;
   cmAlignVisionControllerInterface.configuration.DataConfig.assignableControl.assignable_24 := FALSE;
   cmAlignVisionControllerInterface.configuration.DataConfig.assignableControl.assignable_25 := FALSE;
   cmAlignVisionControllerInterface.configuration.DataConfig.assignableControl.assignable_26 := FALSE;
   cmAlignVisionControllerInterface.configuration.DataConfig.assignableControl.assignable_27 := FALSE;
   cmAlignVisionControllerInterface.configuration.DataConfig.assignableControl.assignable_28 := FALSE;
   cmAlignVisionControllerInterface.configuration.DataConfig.assignableControl.assignable_29 := FALSE;
   cmAlignVisionControllerInterface.configuration.DataConfig.assignableControl.assignable_30 := FALSE;
   cmAlignVisionControllerInterface.configuration.DataConfig.assignableControl.assignable_31 := FALSE;
   cmAlignVisionControllerInterface.configuration.DataConfig.parameterData248Byte_1.reversed0 := 0;
   cmAlignVisionControllerInterface.configuration.DataConfig.parameterData248Byte_1.reserved1 := 0;
   cmAlignVisionControllerInterface.configuration.DataConfig.parameterData248Byte_1.commandNumber := 0;
   cmAlignVisionControllerInterface.configuration.DataConfig.parameterData248Byte_1.cmdParameter[0..15] := 0;
   cmAlignVisionControllerInterface.configuration.DataConfig.parameterData248Byte_1.inDataFieldbus[0..42] := 0;
   cmAlignVisionControllerInterface.configuration.DataConfig.parameterData248Byte_2[0..61] := 0;
   cmAlignVisionControllerInterface.configuration.DataConfig.parameterData248Byte_3[0..61] := 0;
   cmAlignVisionControllerInterface.configuration.DataConfig.parameterData248Byte_4[0..61] := 0;
   cmAlignVisionControllerInterface.configuration.DataConfig.parameterData248Byte_5[0..61] := 0;
   AlignVisionConversion.tabFoldingMissingJudgementResult := 0.0;
   AlignVisionConversion.electrodeLengthJudgementResult := 0.0;
   AlignVisionConversion.electrodeHeightJudgementResult := 0.0;
   AlignVisionConversion.movementAmountAxisX1 := 0.0;
   AlignVisionConversion.movementAmountAxisY1 := 0.0;
   AlignVisionConversion.movementAmountAxisY2 := 0.0;
   AlignVisionConversion.tabFoldingMissingReply := 0.0;
   AlignVisionConversion.tabFoldingMissingUpperRangeReply := 0.0;
   AlignVisionConversion.tabFoldingMissingLowerRangeReply := 0.0;
   AlignVisionConversion.electrodeLengthReply := 0.0;
   AlignVisionConversion.electrodeLengthUpperRangeReply := 0.0;
   AlignVisionConversion.electrodeLengthLowerRangeReply := 0.0;
   AlignVisionConversion.electrodeHeightReply := 0.0;
   AlignVisionConversion.electrodeHeightUpperRangeReply := 0.0;
   AlignVisionConversion.electrodeHeightLowerRangeReply := 0.0;
   AlignVisionHistory.partID[0..50] := '';
   AlignVisionHistory.productionTimestamp[0..50] := DTL#1970-01-01-00:00:00;
   AlignVisionHistory.data[0..50].VisionOk := FALSE;
   AlignVisionHistory.data[0..50].VisionNG := FALSE;
   AlignVisionHistory.data[0..50].VisionComplete := FALSE;
   AlignVisionHistory.data[0..50]."GagueR&Rtype1OK" := FALSE;
   AlignVisionHistory.data[0..50]."GagueR&Rtype1NG" := FALSE;
   AlignVisionHistory.data[0..50]."GagueR&Rtype1Complete" := FALSE;
   AlignVisionHistory.data[0..50]."GagueR&Rtype3OK" := FALSE;
   AlignVisionHistory.data[0..50]."GagueR&Rtype3NG" := FALSE;
   AlignVisionHistory.data[0..50]."GagueR&Rtype3Complete" := FALSE;
   AlignVisionHistory.data[0..50].VisionData.tabFoldingMissingJudgementResult := 0.0;
   AlignVisionHistory.data[0..50].VisionData.electrodeLengthJudgementResult := 0.0;
   AlignVisionHistory.data[0..50].VisionData.electrodeHeightJudgementResult := 0.0;
   AlignVisionHistory.data[0..50].VisionData.movementAmountAxisX1 := 0.0;
   AlignVisionHistory.data[0..50].VisionData.movementAmountAxisY1 := 0.0;
   AlignVisionHistory.data[0..50].VisionData.movementAmountAxisY2 := 0.0;
   AlignVisionHistory.data[0..50].VisionData.tabFoldingMissingReply := 0.0;
   AlignVisionHistory.data[0..50].VisionData.tabFoldingMissingUpperRangeReply := 0.0;
   AlignVisionHistory.data[0..50].VisionData.tabFoldingMissingLowerRangeReply := 0.0;
   AlignVisionHistory.data[0..50].VisionData.electrodeLengthReply := 0.0;
   AlignVisionHistory.data[0..50].VisionData.electrodeLengthUpperRangeReply := 0.0;
   AlignVisionHistory.data[0..50].VisionData.electrodeLengthLowerRangeReply := 0.0;
   AlignVisionHistory.data[0..50].VisionData.electrodeHeightReply := 0.0;
   AlignVisionHistory.data[0..50].VisionData.electrodeHeightUpperRangeReply := 0.0;
   AlignVisionHistory.data[0..50].VisionData.electrodeHeightLowerRangeReply := 0.0;
   intCondition.Axis_07.Home.HomeInterlock := FALSE;
   intCondition.Axis_07.Home.homeinterlock_error := FALSE;
   intCondition.Axis_07.Home.intout[0..9] := FALSE;
   intCondition.Axis_07.Jog.ForwardInterlockOK := FALSE;
   intCondition.Axis_07.Jog.BackwardInterlockOk := FALSE;
   intCondition.Axis_07.Jog.ForwardInterlockError := FALSE;
   intCondition.Axis_07.Jog.BackwardInterlockError := FALSE;
   intCondition.Axis_07.Jog.intOut[0..9] := FALSE;
   intCondition.Axis_07.Position.interlockOk[0..15] := FALSE;
   intCondition.Axis_07.Position.interlockError[0..15] := FALSE;
   intCondition.Axis_07.Position.intOut[0..9] := FALSE;
   intCondition.Axis_08.Home.HomeInterlock := FALSE;
   intCondition.Axis_08.Home.homeinterlock_error := FALSE;
   intCondition.Axis_08.Home.intout[0..9] := FALSE;
   intCondition.Axis_08.Jog.ForwardInterlockOK := FALSE;
   intCondition.Axis_08.Jog.BackwardInterlockOk := FALSE;
   intCondition.Axis_08.Jog.ForwardInterlockError := FALSE;
   intCondition.Axis_08.Jog.BackwardInterlockError := FALSE;
   intCondition.Axis_08.Jog.intOut[0..9] := FALSE;
   intCondition.Axis_08.Position.interlockOk[0..15] := FALSE;
   intCondition.Axis_08.Position.interlockError[0..15] := FALSE;
   intCondition.Axis_08.Position.intOut[0..9] := FALSE;
   intCondition.Axis_09.Home.HomeInterlock := FALSE;
   intCondition.Axis_09.Home.homeinterlock_error := FALSE;
   intCondition.Axis_09.Home.intout[0..9] := FALSE;
   intCondition.Axis_09.Jog.ForwardInterlockOK := FALSE;
   intCondition.Axis_09.Jog.BackwardInterlockOk := FALSE;
   intCondition.Axis_09.Jog.ForwardInterlockError := FALSE;
   intCondition.Axis_09.Jog.BackwardInterlockError := FALSE;
   intCondition.Axis_09.Jog.intOut[0..9] := FALSE;
   intCondition.Axis_09.Position.interlockOk[0..15] := FALSE;
   intCondition.Axis_09.Position.interlockError[0..15] := FALSE;
   intCondition.Axis_09.Position.intOut[0..9] := FALSE;
   intCondition.Axis_10.Home.HomeInterlock := FALSE;
   intCondition.Axis_10.Home.homeinterlock_error := FALSE;
   intCondition.Axis_10.Home.intout[0..9] := FALSE;
   intCondition.Axis_10.Jog.ForwardInterlockOK := FALSE;
   intCondition.Axis_10.Jog.BackwardInterlockOk := FALSE;
   intCondition.Axis_10.Jog.ForwardInterlockError := FALSE;
   intCondition.Axis_10.Jog.BackwardInterlockError := FALSE;
   intCondition.Axis_10.Jog.intOut[0..9] := FALSE;
   intCondition.Axis_10.Position.interlockOk[0..15] := FALSE;
   intCondition.Axis_10.Position.interlockError[0..15] := FALSE;
   intCondition.Axis_10.Position.intOut[0..9] := FALSE;
   intCondition.Axis_13.Home.HomeInterlock := FALSE;
   intCondition.Axis_13.Home.homeinterlock_error := FALSE;
   intCondition.Axis_13.Home.intout[0..9] := FALSE;
   intCondition.Axis_13.Jog.ForwardInterlockOK := FALSE;
   intCondition.Axis_13.Jog.BackwardInterlockOk := FALSE;
   intCondition.Axis_13.Jog.ForwardInterlockError := FALSE;
   intCondition.Axis_13.Jog.BackwardInterlockError := FALSE;
   intCondition.Axis_13.Jog.intOut[0..9] := FALSE;
   intCondition.Axis_13.Position.interlockOk[0..15] := FALSE;
   intCondition.Axis_13.Position.interlockError[0..15] := FALSE;
   intCondition.Axis_13.Position.intOut[0..9] := FALSE;
   intCondition.Axis_18.Home.HomeInterlock := FALSE;
   intCondition.Axis_18.Home.homeinterlock_error := FALSE;
   intCondition.Axis_18.Home.intout[0..9] := FALSE;
   intCondition.Axis_18.Jog.ForwardInterlockOK := FALSE;
   intCondition.Axis_18.Jog.BackwardInterlockOk := FALSE;
   intCondition.Axis_18.Jog.ForwardInterlockError := FALSE;
   intCondition.Axis_18.Jog.BackwardInterlockError := FALSE;
   intCondition.Axis_18.Jog.intOut[0..9] := FALSE;
   intCondition.Axis_18.Position.interlockOk[0..15] := FALSE;
   intCondition.Axis_18.Position.interlockError[0..15] := FALSE;
   intCondition.Axis_18.Position.intOut[0..9] := FALSE;
   intCondition.Axis_19.Home.HomeInterlock := FALSE;
   intCondition.Axis_19.Home.homeinterlock_error := FALSE;
   intCondition.Axis_19.Home.intout[0..9] := FALSE;
   intCondition.Axis_19.Jog.ForwardInterlockOK := FALSE;
   intCondition.Axis_19.Jog.BackwardInterlockOk := FALSE;
   intCondition.Axis_19.Jog.ForwardInterlockError := FALSE;
   intCondition.Axis_19.Jog.BackwardInterlockError := FALSE;
   intCondition.Axis_19.Jog.intOut[0..9] := FALSE;
   intCondition.Axis_19.Position.interlockOk[0..15] := FALSE;
   intCondition.Axis_19.Position.interlockError[0..15] := FALSE;
   intCondition.Axis_19.Position.intOut[0..9] := FALSE;
   intCondition.Axis_20.Home.HomeInterlock := FALSE;
   intCondition.Axis_20.Home.homeinterlock_error := FALSE;
   intCondition.Axis_20.Home.intout[0..9] := FALSE;
   intCondition.Axis_20.Jog.ForwardInterlockOK := FALSE;
   intCondition.Axis_20.Jog.BackwardInterlockOk := FALSE;
   intCondition.Axis_20.Jog.ForwardInterlockError := FALSE;
   intCondition.Axis_20.Jog.BackwardInterlockError := FALSE;
   intCondition.Axis_20.Jog.intOut[0..9] := FALSE;
   intCondition.Axis_20.Position.interlockOk[0..15] := FALSE;
   intCondition.Axis_20.Position.interlockError[0..15] := FALSE;
   intCondition.Axis_20.Position.intOut[0..9] := FALSE;
   intCondition.Actuator_23.Home_INT := FALSE;
   intCondition.Actuator_23.Work_INT := FALSE;
   intCondition.Actuator_23.Home_INT_Error := FALSE;
   intCondition.Actuator_23.Work_INT_Error := FALSE;
   intCondition.Actuator_23.intOut[0..9] := FALSE;
   intCondition.Actuator_24.Home_INT := FALSE;
   intCondition.Actuator_24.Work_INT := FALSE;
   intCondition.Actuator_24.Home_INT_Error := FALSE;
   intCondition.Actuator_24.Work_INT_Error := FALSE;
   intCondition.Actuator_24.intOut[0..9] := FALSE;
   intCondition.Actuator_25.Home_INT := FALSE;
   intCondition.Actuator_25.Work_INT := FALSE;
   intCondition.Actuator_25.Home_INT_Error := FALSE;
   intCondition.Actuator_25.Work_INT_Error := FALSE;
   intCondition.Actuator_25.intOut[0..9] := FALSE;
   intCondition.Actuator_26.Home_INT := FALSE;
   intCondition.Actuator_26.Work_INT := FALSE;
   intCondition.Actuator_26.Home_INT_Error := FALSE;
   intCondition.Actuator_26.Work_INT_Error := FALSE;
   intCondition.Actuator_26.intOut[0..9] := FALSE;
   intCondition.Actuator_27.Home_INT := FALSE;
   intCondition.Actuator_27.Work_INT := FALSE;
   intCondition.Actuator_27.Home_INT_Error := FALSE;
   intCondition.Actuator_27.Work_INT_Error := FALSE;
   intCondition.Actuator_27.intOut[0..9] := FALSE;
   intCondition.Actuator_28.Home_INT := FALSE;
   intCondition.Actuator_28.Work_INT := FALSE;
   intCondition.Actuator_28.Home_INT_Error := FALSE;
   intCondition.Actuator_28.Work_INT_Error := FALSE;
   intCondition.Actuator_28.intOut[0..9] := FALSE;
   intCondition.Actuator_29.Home_INT := FALSE;
   intCondition.Actuator_29.Work_INT := FALSE;
   intCondition.Actuator_29.Home_INT_Error := FALSE;
   intCondition.Actuator_29.Work_INT_Error := FALSE;
   intCondition.Actuator_29.intOut[0..9] := FALSE;
   intCondition.Actuator_30.Home_INT := FALSE;
   intCondition.Actuator_30.Work_INT := FALSE;
   intCondition.Actuator_30.Home_INT_Error := FALSE;
   intCondition.Actuator_30.Work_INT_Error := FALSE;
   intCondition.Actuator_30.intOut[0..9] := FALSE;
   intCondition.Actuator_31.Home_INT := FALSE;
   intCondition.Actuator_31.Work_INT := FALSE;
   intCondition.Actuator_31.Home_INT_Error := FALSE;
   intCondition.Actuator_31.Work_INT_Error := FALSE;
   intCondition.Actuator_31.intOut[0..9] := FALSE;
   intCondition.Actuator_32.Home_INT := FALSE;
   intCondition.Actuator_32.Work_INT := FALSE;
   intCondition.Actuator_32.Home_INT_Error := FALSE;
   intCondition.Actuator_32.Work_INT_Error := FALSE;
   intCondition.Actuator_32.intOut[0..9] := FALSE;
END_DATA_BLOCK
